FUNCTION_BLOCK FB_ConsoleLogger IMPLEMENTS  I_Logger

VAR
END_VAR

{warning 'add method implementation '}
METHOD M_Log : BOOL
VAR_INPUT
	sMessage	: STRING(255);
END_VAR

ADSLOGSTR(msgCtrlMask:= ADSLOG_MSGTYPE_ERROR,
			msgFmtStr := 'Console log: %s',
			strArg := sMessage);
END_METHOD

END_FUNCTION_BLOCK

(* stored: Version 1.1.0.1, ProductVersion 3.1.4024.16
   POU FB_ConsoleLogger: Id {50349c97-3a06-4359-b976-d357416472e3}, SpecialFunc None
   Method M_Log: Id {c9bee7fa-eb16-44ec-81ae-589c1b94fb65} *)
